Yaskawa INFORM job: FORLOOPTEST0311.JBI

/JOB
//NAME FORLOOPTEST
//POS
///NPOS 3,0,0,0,0,0
///TOOL 5
///POSTYPE PULSE
///PULSE
C00000=-3,-50477,-58433,3,-74931,486
C00001=-21533,13564,-68096,-82219,-30330,47469
C00002=-3,-50477,-58433,3,-74931,486
//INST
///DATE 2024/03/11 14:13
///COMM For loop test
///ATTR SC,RW
///GROUP1 RB1
NOP
MOVJ C00000 VJ=3.00
MOVJ C00001 VJ=2.00
FOR I001 START= 0 TO 2
	 FOR I000 START= 2 TO 3
		 MOVL P[I000] V=I[I000]
	 NEXT I000
NEXT I001
MOVJ C00002 VJ=3.00
END
